// TIA Portal V20 export
// export: Created 2025-12-01T14:57:16.4603031Z, ExportSetting None, DisplayName Totally Integrated Automation Portal, DisplayVersion V20 Update 3, DisplayName TIA Portal Openness, DisplayVersion V20 Update 3, DisplayName TIA Portal Version Control Interface, DisplayVersion V20 Update 3, DisplayName STEP 7 Professional, DisplayVersion V20 Update 3, DisplayName STEP 7 Safety, DisplayVersion V20 Update 2, DisplayName WinCC Basic/Comfort/Advanced, DisplayVersion V20 Update 3, DisplayName WinCC Professional, DisplayVersion V20 Update 3, DisplayName WinCC Unified, DisplayVersion V20 Update 3
DATA_BLOCK "DB861_FIFO_Errores"   // DB861
{ S7_Optimized_Access := 'FALSE' }
AUTHOR : ERRORES
NAME : 20131009
VERSION : 3.1
// stored: AutoNumber false
   VAR
      IndiceExtracion : UInt;   // Indice de visualización de Errores
      ArmariosGraves : Array[0.."CTE_MaxDispositivos"] of UDInt;   // Codigo de Error Grave de los Dispositivos (CCPIF uy CBOX's)
      ArmariosLeves : Array[0.."CTE_MaxDispositivos"] of UDInt;   // Codigo de Error Leve de los Dispositivos (CCPIF uy CBOX's)
      Mesas : Array[0.."CTE_MaxMesas"] of UDInt;   // Codigo de Error de las Mesas
      Maquinas : Array[0.."CTE_MaxMesas"] of UDInt;   // Codigo de Error de las Maquinas
      Final : UDInt;
   END_VAR
BEGIN
END_DATA_BLOCK
